// TIA Portal V17 export
// export: Created 2025-03-05T08:02:58.862828Z, ExportSetting WithDefaults, DisplayName Totally Integrated Automation Portal, DisplayVersion V17 Update 8, DisplayName TIA Portal Openness, DisplayVersion V17 Update 8, DisplayName TIA Portal Version Control Interface, DisplayVersion V17, DisplayName SINAMICS Startdrive Advanced, DisplayVersion V17 SP2, DisplayName SINAMICS Startdrive G110M, G120, G120C, G120D, G120P, G115D, DisplayVersion V17 SP2, DisplayName SINAMICS Startdrive G130, G150, S120, S150, SINAMICS MV, S210, DisplayVersion V17 SP2, DisplayName STEP 7 Professional, DisplayVersion V17 Update 8, DisplayName SINUMERIK ONE STEP 7 Toolbox, DisplayVersion V17 Update 12, DisplayName SINUMERIK 840D sl STEP 7 Toolbox, DisplayVersion V17 Update 12, DisplayName STEP 7 Safety, DisplayVersion V17 Update 6, DisplayName WinCC Advanced, DisplayVersion V17 Update 8
FUNCTION_BLOCK "FB16700_POWDER_FLOW_DATA_SAVE"   // FB16700, LAD
{ S7_Optimized_Access := 'TRUE' }
VERSION : 0.1
// stored: AutoNumber false, IsIECCheckEnabled false, IsRetainMemResEnabled false, MemoryReserve 100, SetENOAutomatically false, UDAEnableTagReadback false
   VAR_INPUT
      iMEDICOAT_DATA : Int;
   END_VAR
   VAR_OUTPUT
      oMEDICOAT_DATA_ARRAY : Array[1..20] of "MEDICOAT_TIME_STAMP";
   END_VAR
   VAR_IN_OUT
      ARRAY_NUMBER_MEMORY : Int := 1;
   END_VAR
   VAR
      SAVE_VALUE_TRIGGER_TON : TON_TIME;
      RESET_VALUE_TON { S7_SetPoint := 'True'} : TON_TIME;
      SAVE_VALUE_TRIGGER { S7_SetPoint := 'True'} : Bool;
      RESET_TIMER_AUX : Bool;
      PULSE_AUX : Bool;
   END_VAR
   VAR_TEMP
      TIME_READ_RET_VAL : Int;
      ARRAY_MEMORY_AUX : Int;
   END_VAR
   VAR_TEMP   // added for the SCL form of the ladder/FBD networks
      _w1 : Bool;
   END_VAR
BEGIN

REGION Network 1
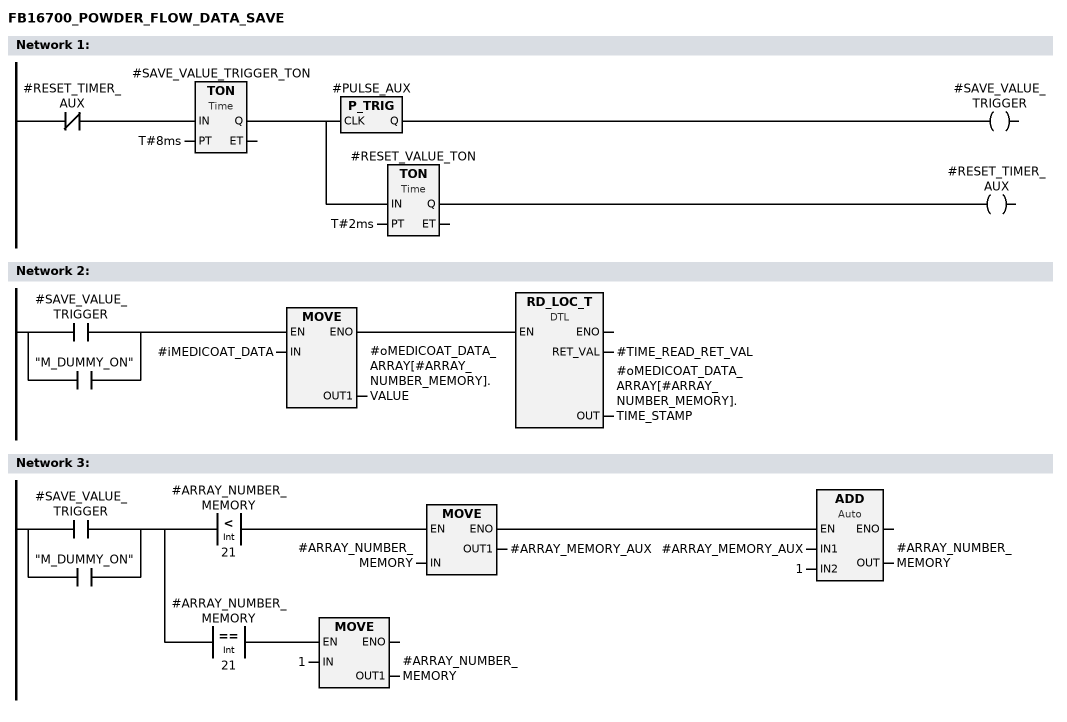
   RUNG wire#powerrail
      I_Contact( #RESET_TIMER_AUX )
      { S7_Templates := "time_type := Time" } #SAVE_VALUE_TRIGGER_TON.TON(pt := T#8ms, et =>)
      wire#w1
      P_Trig( #PULSE_AUX )
      Coil( #SAVE_VALUE_TRIGGER )
   END_RUNG
   RUNG wire#w1
      { S7_Templates := "time_type := Time" } #RESET_VALUE_TON.TON(pt := T#2ms, et =>)
      Coil( #RESET_TIMER_AUX )
   END_RUNG
   // the same network as SCL:
   #SAVE_VALUE_TRIGGER_TON(IN := NOT #RESET_TIMER_AUX, PT := T#8ms);   // TON
   #_w1 := #SAVE_VALUE_TRIGGER_TON.Q AND NOT #PULSE_AUX;   // rising edge
   #PULSE_AUX := #SAVE_VALUE_TRIGGER_TON.Q;
   #SAVE_VALUE_TRIGGER := #_w1;
   #RESET_VALUE_TON(IN := #SAVE_VALUE_TRIGGER_TON.Q, PT := T#2ms);   // TON
   #RESET_TIMER_AUX := #RESET_VALUE_TON.Q;
END_REGION

REGION Network 2
   RUNG wire#powerrail
      Contact( #SAVE_VALUE_TRIGGER )
      wire#w1
      Move(in := #iMEDICOAT_DATA, out1 => #oMEDICOAT_DATA_ARRAY[#ARRAY_NUMBER_MEMORY].VALUE)
      { S7_Templates := "date_type := DTL" } RD_LOC_T(RET_VAL => #TIME_READ_RET_VAL, OUT => #oMEDICOAT_DATA_ARRAY[#ARRAY_NUMBER_MEMORY].TIME_STAMP)
   END_RUNG
   RUNG wire#powerrail
      Contact( "M_DUMMY_ON" )
   END_RUNG wire#w1
   // the same network as SCL:
   IF #SAVE_VALUE_TRIGGER OR "M_DUMMY_ON" THEN
       #oMEDICOAT_DATA_ARRAY[#ARRAY_NUMBER_MEMORY].VALUE := #iMEDICOAT_DATA;
       #TIME_READ_RET_VAL := RD_LOC_T(OUT => #oMEDICOAT_DATA_ARRAY[#ARRAY_NUMBER_MEMORY].TIME_STAMP);
   END_IF;
END_REGION

REGION Network 3
   RUNG wire#powerrail
      Contact( #SAVE_VALUE_TRIGGER )
      wire#w1
      { S7_Templates := "SrcType := Int" } LT_Contact(in1 := #ARRAY_NUMBER_MEMORY, in2 := 21)
      Move(in := #ARRAY_NUMBER_MEMORY, out1 => #ARRAY_MEMORY_AUX)
      Add(in1 := #ARRAY_MEMORY_AUX, in2 := 1, out => #ARRAY_NUMBER_MEMORY)
   END_RUNG
   RUNG wire#powerrail
      Contact( "M_DUMMY_ON" )
   END_RUNG wire#w1
   RUNG wire#w1
      { S7_Templates := "SrcType := Int" } EQ_Contact(in1 := #ARRAY_NUMBER_MEMORY, in2 := 21)
      Move(in := 1, out1 => #ARRAY_NUMBER_MEMORY)
   END_RUNG
   // the same network as SCL:
   #_w1 := #SAVE_VALUE_TRIGGER OR "M_DUMMY_ON";
   IF #_w1 AND (#ARRAY_NUMBER_MEMORY < 21) THEN
       #ARRAY_MEMORY_AUX := #ARRAY_NUMBER_MEMORY;
       #ARRAY_NUMBER_MEMORY := #ARRAY_MEMORY_AUX + 1;
   END_IF;
   IF #_w1 AND (#ARRAY_NUMBER_MEMORY = 21) THEN #ARRAY_NUMBER_MEMORY := 1; END_IF;
END_REGION
END_FUNCTION_BLOCK
